// TIA Portal V16 export
// export: Created 2024-09-05T15:58:42.5352565Z, ExportSetting WithDefaults, DisplayName Totally Integrated Automation Portal, DisplayVersion V16 Update 6, DisplayName TIA Portal Version Control Interface, DisplayVersion V16 Update 2, DisplayName TIA Portal Openness, DisplayVersion V16 Update 6, DisplayName STEP 7 Professional, DisplayVersion V16 Update 6, DisplayName STEP 7 Safety, DisplayVersion V16, DisplayName WinCC Advanced, DisplayVersion V16 Update 6
VAR_GLOBAL   // PLC tag table "R1"
   qR1drivesOn AT %Q800.0 : Bool;
   qR1confMess AT %Q800.1 : Bool;
   qR1ExtStart AT %Q800.2 : Bool;
   qR1moveEnable AT %Q800.3 : Bool;
   qR1reqHome AT %Q800.6 : Bool;
   qR1pgNoValid AT %Q800.7 : Bool;
   qR1reqDoor AT %Q801.0 : Bool;
   qR1jobNr AT %QB802 : Byte;
   qR1_MM220grippingTubeInBp AT %Q804.0 : Bool;
   qR1_MM220grippingTubeInWp AT %Q804.1 : Bool;
   qR1_MM222holdingSidememberInsideInBp AT %Q804.2 : Bool;
   qR1_MM222holdingSidememberInsideInWp AT %Q804.3 : Bool;
   iR1periReady AT %I800.0 : Bool;
   iR1stopMess AT %I800.1 : Bool;
   iR1progAct AT %I800.2 : Bool;
   iR1onPath AT %I800.3 : Bool;
   iR1ext AT %I800.4 : Bool;
   iR1internalEstop AT %I800.5 : Bool;
   iR1home AT %I800.6 : Bool;
   iR1pgNoReq AT %I800.7 : Bool;
   iR1robStopped AT %I801.0 : Bool;
   iR1jobNr AT %IB802 : Byte;
   iR1_MM220grippingTubeToBp AT %I804.0 : Bool;
   iR1_MM220grippingTubeToWp AT %I804.1 : Bool;
   iR1_MM222holdingSidememberInsideToBp AT %I804.2 : Bool;
   iR1_MM222holdingSidememberInsideToWp AT %I804.3 : Bool;
   iR1inPickupStartPositionSt2 AT %I804.6 : Bool;
   iR1outOf_AE_left_bottom AT %I854.3 : Bool;   // autoeject left
   iR1PartReleased AT %I804.4 : Bool;
   iR1PartInGripper AT %I804.5 : Bool;
   iR1err1 AT %I809.0 : Bool;
   iR1err2 AT %I809.1 : Bool;
   iR1err3 AT %I809.2 : Bool;
   iR1err4 AT %I809.3 : Bool;
   iR1err5 AT %I809.4 : Bool;
   iR1err6 AT %I809.5 : Bool;
   iR1err7 AT %I809.6 : Bool;
   iR1err8 AT %I809.7 : Bool;
   iR1OutOfSt2 AT %I854.0 : Bool;   // carousel
   iR1ActionRunning AT %I801.2 : Bool;
   iR1OutOfSt3 AT %I854.1 : Bool;   // jig
   qR1BreaktestReq AT %Q805.1 : Bool;
   qR1MasteringReq AT %Q805.0 : Bool;
   iR1_MM224holdingSidememberOutsideToBp AT %I805.3 : Bool;
   iR1_MM224holdingSidememberOutsideToWp AT %I805.4 : Bool;
   qR1_MM224holdingSidememberOutsideInBp AT %Q804.5 : Bool;
   qR1_MM224holdingSidememberOutsideInWp AT %Q804.6 : Bool;
   qR1NHE AT %Q850.1 : Bool;   // safety for manual
   qR1BS1 AT %Q850.2 : Bool;   // safety for auto
   qR1BS2 AT %Q850.3 : Bool;   // safety for auto
   qR1SHS1 AT %Q850.4 : Bool;   // safety for manual
   qR1SHS2 AT %Q850.5 : Bool;   // safety for manual
   qR1SBH AT %Q851.1 : Bool;   // safety for manual
   iR1EmgOK_NHL AT %I850.0 : Bool;
   iR1OutOfSt4 AT %I854.2 : Bool;   // hanger manipulator
   qR1ToolSelect1 AT %Q856.0 : Bool;
   qR1ToolSelect2 AT %Q856.1 : Bool;
   iR1rearInWorkZone1 AT %I854.7 : Bool;
   iR1rearInWorkZone2 AT %I855.0 : Bool;
   iR1rearInWorkZone3 AT %I855.1 : Bool;
   qR1_ST3free AT %Q804.7 : Bool;
   iR1masteringReq AT %I806.0 : Bool;
   iR1braktestReq AT %I806.1 : Bool;
   qR1frontTubePresent AT %Q805.2 : Bool;
   qR1rearTubePresent AT %Q805.3 : Bool;
   qR1typeRH AT %Q805.4 : Bool;
   iR1outOf_AE_right_bottom AT %I854.4 : Bool;   // autoeject right
   iR1inDropoffStartPositionSt3 AT %I805.2 : Bool;
   iR1inSt3 AT %I804.7 : Bool;
   iR1inPickupStartPositionAutoeject AT %I805.5 : Bool;
   iR1outOf_AE_left_top AT %I854.5 : Bool;
   iR1outOf_AE_right_top AT %I854.6 : Bool;
   iR1inDropoffStartPositionHanger AT %I805.6 : Bool;
   iR1deadmanSwitch AT %I850.3 : Bool;
END_VAR
